Fanuc KAREL source: IO0076.KL

-- PROVISIONAL review KL for V770-1; original PC SHA256 8c8fbe215b46b7a07b0f71b881d1d24fa7e9d9f6adf90e3e40f40c3c68f67265
-- Incomplete behavior may be omitted. Consult companion uncertainty JSON. Do not deploy.
PROGRAM IO0076
%NOLOCKGROUP
-- UNRESOLVED_LOCAL_POOL 5 cells at code offset 13; source declarations unknown
-- DIRECT_LOCAL_WORD_ACCESS alone does not prove INTEGER, REAL, or BOOLEAN
BEGIN
  -- UNRESOLVED_PC offsets 0-18; opcodes 2B,2C,7B
  -- UNRESOLVED_PC offsets 23-30; opcodes 9D,23
  -- UNRESOLVED_PC offsets 35-49; opcodes 2E,22,9D,33,35
  -- UNRESOLVED_PC offsets 54-61; opcodes 9D,23
  -- UNRESOLVED_PC offsets 66-77; opcodes 2E,23
  -- UNRESOLVED_PC offsets 82-92; opcodes 9D,19,64,23
  -- UNRESOLVED_PC offsets 97-101; opcodes 7F
  -- UNRESOLVED_PC offsets 106-110; opcodes 27,AA
  -- UNRESOLVED_PC offsets 115-119; opcodes 7F
END IO0076
